FUNCTION_BLOCK repaint (* Basic Function Block Type *)
  (* Standard: 61499-2 *)
  (* Version 0.0, 2006-01-11, Anirudha, UoA *)
  (* Compiler header: package fb.rt.vhmi; *)
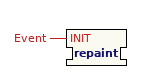
  EVENT_INPUT
    INIT; (* Initialization Request *)
  END_EVENT
END_FUNCTION_BLOCK
